KUKA KRL data list: ap_1.dat

&ACCESS RVP
&REL 15
&PARAM EDITMASK = *
&PARAM TEMPLATE = C:\KRC\Roboter\Template\ExpertVorgabe
&PARAM DISKPATH = KRC:\R1\Program
DEFDAT  ap_1
DECL E6POS XP1={X 170.668137,Y 87.8043442,Z 190.158340,A 179.701111,B 5.22395840E-06,C -5.58706188E-06,S 2,T 35,E1 0.0,E2 0.0,E3 0.0,E4 0.0,E5 0.0,E6 0.0}
DECL FDAT FP1={TOOL_NO 1,BASE_NO 1,IPO_FRAME #BASE,POINT2[] " "}
DECL PDAT PPDAT1={VEL 50.0000,ACC 50.0000,APO_DIST 500.000,APO_MODE #CDIS,GEAR_JERK 100.000,EXAX_IGN 0}
DECL MODULEPARAM_T LAST_TP_PARAMS={PARAMS[] "Kuka.PointName=P4; Kuka.FrameData.base_no=1; Kuka.FrameData.tool_no=1; Kuka.FrameData.ipo_frame=#BASE; Kuka.FrameData.point2=; Kuka.isglobalpoint=False; Kuka.MoveDataPtpName=PDAT3; Kuka.MovementDataPdat.apo_mode=#CDIS; Kuka.MovementDataPdat.apo_dist=500; Kuka.MovementData.vel=0.01; Kuka.MovementData.acc=50; Kuka.MovementData.exax_ign=0; Kuka.VelocityPtp=50; Kuka.BlendingEnabled=False; Kuka.APXEnabled=False; Kuka.CurrentCDSetIndex=0; Kuka.MoveDataName=CPDAT2; Kuka.MovementData.cb={AUX_PT {ORI #CONSIDER,E1 #CONSIDER,E2 #CONSIDER,E3 #CONSIDER,E4 #CONSIDER,E5 #CONSIDER,E6 #CONSIDER},TARGET_PT {ORI #INTERPOLATE,E1 #INTERPOLATE,E2 #INTERPOLATE,E3 #INTERPOLATE,E4 #INTERPOLATE,E5 #INTERPOLATE,E6 #INTERPOLATE}}; Kuka.MovementData.apo_fac=50; Kuka.MovementData.apo_dist=50; Kuka.MovementData.axis_acc=100; Kuka.MovementData.axis_vel=100; Kuka.MovementData.circ_typ=#BASE; Kuka.MovementData.jerk_fac=50; Kuka.MovementData.ori_typ=#VAR; Kuka.VelocityPath=0.01; ArcTech.WdatVarName=WDAT2                                                   "}
DECL E6POS XP2={X 44.5445099,Y 61.0237160,Z 5.54459429,A 179.701111,B 5.32584318E-06,C -5.64468837E-06,S 2,T 35,E1 0.0,E2 0.0,E3 0.0,E4 0.0,E5 0.0,E6 0.0}
DECL FDAT FP2={TOOL_NO 1,BASE_NO 1,IPO_FRAME #BASE,POINT2[] " "}
DECL PDAT PPDAT2={VEL 100.000,ACC 50.0000,APO_DIST 500.000,APO_MODE #CDIS,GEAR_JERK 100.000,EXAX_IGN 0}
DECL stArcDat_T WDAT1={WdatId[] "WDAT1",Strike {JobModeId[] "Job mode",StartTime 0.0,PreFlowTime 0.0,Channel1 0.0,Channel2 0.0,Channel3 0.0,Channel4 0.0,Channel5 0.0,Channel6 0.0,Channel7 0.0,Channel8 0.0,PurgeTime 0.0},Weld {JobModeId[] "Job mode",ParamSetId[] "Set1",Velocity 0.00416666688,Channel1 13.0000,Channel2 0.0,Channel3 0.0,Channel4 0.0,Channel5 0.0,Channel6 0.0,Channel7 0.0,Channel8 0.0},Weave {Pattern #Trapecoid,Length 2.00000,Amplitude 6.00000,Angle 90.0000,LeftSideDelay 0.0,RightSideDelay 0.0}}
DECL stArcDat_T WP3={WdatId[] "WP3",Info {Version 304031264},Strike {SeamName[] " ",PartName[] " ",SeamNumber 0,PartNumber 0,DesiredLength 0.0,LengthTolNeg 0.0,LengthTolPos 0.0,LengthCtrlActive FALSE}}
DECL E6POS XP3={X 17.3123798,Y 74.5600,Z -8.14224339,A 179.701111,B 5.31830847E-06,C -5.68684300E-06,S 2,T 35,E1 0.0,E2 0.0,E3 0.0,E4 0.0,E5 0.0,E6 0.0}
DECL FDAT FP3={TOOL_NO 1,BASE_NO 1,IPO_FRAME #BASE,POINT2[] " "}
DECL LDAT LCPDAT1={VEL 0.500000,ACC 50.0000,APO_DIST 50.0000,APO_FAC 50.0000,AXIS_VEL 100.000,AXIS_ACC 100.000,ORI_TYP #VAR,CIRC_TYP #BASE,JERK_FAC 50.0000,GEAR_JERK 100.000,EXAX_IGN 0,CB {AUX_PT {ORI #CONSIDER,E1 #CONSIDER,E2 #CONSIDER,E3 #CONSIDER,E4 #CONSIDER,E5 #CONSIDER,E6 #CONSIDER},TARGET_PT {ORI #INTERPOLATE,E1 #INTERPOLATE,E2 #INTERPOLATE,E3 #INTERPOLATE,E4 #INTERPOLATE,E5 #INTERPOLATE,E6 #INTERPOLATE}}}
DECL stArcDat_T WDAT2={WdatId[] "WDAT2",Crater {JobModeId[] "Job mode",ParamSetId[] "Set2",CraterTime 0.500000,PostflowTime 2.00000,Channel1 13.0000,Channel2 0.0,Channel3 0.0,Channel4 0.0,Channel5 0.0,Channel6 0.0,Channel7 0.0,Channel8 0.0,BurnBackTime 0.0}}
DECL stArcDat_T WP4={WdatId[] "WP4",Info {Version 304031264}}
DECL E6POS XP4={X 198.320389,Y 74.5600,Z -8.14224243,A 179.701111,B 5.32127115E-06,C -5.69861913E-06,S 2,T 35,E1 0.0,E2 0.0,E3 0.0,E4 0.0,E5 0.0,E6 0.0}
DECL FDAT FP4={TOOL_NO 1,BASE_NO 1,IPO_FRAME #BASE,POINT2[] " "}
DECL LDAT LCPDAT2={VEL 0.01000000,ACC 50.0000,APO_DIST 50.0000,APO_FAC 50.0000,AXIS_VEL 100.000,AXIS_ACC 100.000,ORI_TYP #VAR,CIRC_TYP #BASE,JERK_FAC 50.0000,GEAR_JERK 100.000,EXAX_IGN 0,CB {AUX_PT {ORI #CONSIDER,E1 #CONSIDER,E2 #CONSIDER,E3 #CONSIDER,E4 #CONSIDER,E5 #CONSIDER,E6 #CONSIDER},TARGET_PT {ORI #INTERPOLATE,E1 #INTERPOLATE,E2 #INTERPOLATE,E3 #INTERPOLATE,E4 #INTERPOLATE,E5 #INTERPOLATE,E6 #INTERPOLATE}}}
DECL E6POS XP5={X 182.544754,Y 74.1202316,Z 135.508194,A 179.701111,B 5.32868034E-06,C -5.65961591E-06,S 2,T 35,E1 0.0,E2 0.0,E3 0.0,E4 0.0,E5 0.0,E6 0.0}
DECL FDAT FP5={TOOL_NO 1,BASE_NO 1,IPO_FRAME #BASE,POINT2[] " "}
DECL PDAT PPDAT3={VEL 50.0000,ACC 50.0000,APO_DIST 500.000,APO_MODE #CDIS,GEAR_JERK 100.000,EXAX_IGN 0}
ENDDAT
